TYPE stHugeArrayOfPrimitive :
STRUCT
	// 1,024 BYTES
	arr_of_primitive : ARRAY[0..1023] OF BYTE;
END_STRUCT
END_TYPE

(* stored: Version 1.1.0.1, ProductVersion 3.1.4024.6
   DUT stHugeArrayOfPrimitive: Id {40fb820d-7397-40e2-bb24-1cce1deef77e} *)
